FUNCTION Convert_USINT_TO_LWORD : Hresult
VAR_INPUT
	in : USINT;
	out : REFERENCE TO LWORD;
END_VAR
VAR
	converted : LWORD;
END_VAR
VAR CONSTANT
	INCOMPATIBLE : HRESULT := 16#9811070E;
END_VAR

converted := USINT_TO_LWORD(in);

IF (LWORD_TO_USINT(converted) <> in) THEN
	Convert_USINT_TO_LWORD := INCOMPATIBLE;
	RETURN;
END_IF

out := converted;

END_FUNCTION

(* stored: Version 1.1.0.1, ProductVersion 3.1.4024.12
   POU Convert_USINT_TO_LWORD: Id {4f8dcf67-da67-4cf2-b841-78f7c50167fb}, SpecialFunc None *)
